// TIA Portal project "Elevator_V16" (V16)

(* hardware
DEVICE "S7-1200 station_1"  S7-1200 Station
   slot 0: "Rack_0"  S7-1200 Rack  Rack  V1.0
   slot 1: "PLC_1"  CPU 1217C DC/DC/DC  6ES7 217-1AG40-0XB0  V4.2
DEVICE "HMI_1"  KTP700 Basic PN
   slot 0: "KTP700 Basic PN"  KTP700 Basic PN  6AV2 123-2GB03-0AX0  14.0.1.0
   slot 1: "HMI_RT_1"  KTP700 Basic PN  6AV2 123-2GB03-0AX0  14.0.1.0
   slot 5: "HMI_1.IE_CP_1"  PROFINET Interface  14.0.1.0
      slot 1: "PROFINET Interface_1"  PROFINET Interface
         slot 1: "Port_1"  Port
*)

// ===== PLC "PLC_1"  CPU 1217C DC/DC/DC =====

VAR_GLOBAL   // PLC tag table "Default tag table"
   "Tag_1" AT %M20.0 : Bool;
END_VAR

DATA_BLOCK "DB_Main"   // DB1
{ S7_Optimized_Access := 'TRUE' }
VERSION : 0.1
   VAR
      Floor1 : Struct
         Request_PB : Bool;
         OpenDoor : Bool;
         OpenDoor_Timer : TON_TIME;
         OneShot_1 : Bool;
      END_STRUCT;
      Floor2 : Struct
         Request_PB : Bool;
         OpenDoor : Bool;
         OpenDoor_Timer : TON_TIME;
         OneShot_1 : Bool;
      END_STRUCT;
      Floor3 : Struct
         Request_PB : Bool;
         OpenDoor : Bool;
         OpenDoor_Timer : TON_TIME;
         OneShot_1 : Bool;
      END_STRUCT;
      Elevator : Struct
         Floor1_PB : Bool;
         Floor2_PB : Bool;
         Floor3_PB : Bool;
         Floor1_Scheduled : Bool;
         Floor2_Scheduled : Bool;
         Floor3_Scheduled : Bool;
         At_Floor1 : Bool;
         At_Floor2 : Bool;
         At_Floor3 : Bool;
         CurrentFloor : Int;
         NextFloorToService : Int;
         Motor_CW : Bool;
         Motor_CCW : Bool;
         GoingUp_Timer_1 : TON_TIME;
         GoingUp_Timer_2 : TON_TIME;
         GoingDown_Timer1 : TON_TIME;
         GoingDown_Timer2 : TON_TIME;
         OneShot_1 : Bool;
         OneShot_2 : Bool;
      END_STRUCT;
   END_VAR
BEGIN
END_DATA_BLOCK

ORGANIZATION_BLOCK "Main"   // OB1, LAD, ProgramCycle
TITLE = "Main Program Sweep (Cycle)"
{ S7_Optimized_Access := 'TRUE' }
VERSION : 0.1
   VAR_INPUT
      Initial_Call : Bool;   // Initial call of this OB
      Remanence : Bool;   // =True, if remanent data are available
   END_VAR
   VAR_TEMP   // added for the SCL form of the ladder/FBD networks
      _w1 : Bool;
      _w2 : Bool;
      _w3 : Bool;
      _w4 : Bool;
      _w5 : Bool;
      _w6 : Bool;
   END_VAR
BEGIN

REGION Network 1: Mange Scheduled Floors
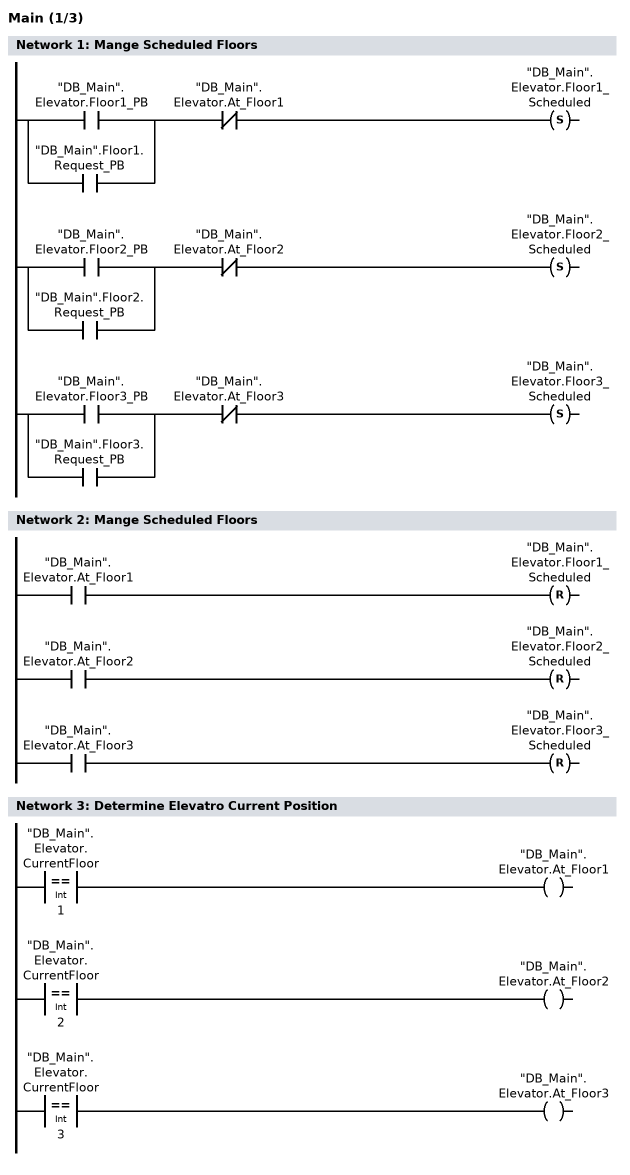
   RUNG wire#powerrail
      Contact( "DB_Main".Elevator.Floor1_PB )
      wire#w1
      I_Contact( "DB_Main".Elevator.At_Floor1 )
      S_Coil( "DB_Main".Elevator.Floor1_Scheduled )
   END_RUNG
   RUNG wire#powerrail
      Contact( "DB_Main".Floor1.Request_PB )
   END_RUNG wire#w1
   RUNG wire#powerrail
      Contact( "DB_Main".Elevator.Floor2_PB )
      wire#w2
      I_Contact( "DB_Main".Elevator.At_Floor2 )
      S_Coil( "DB_Main".Elevator.Floor2_Scheduled )
   END_RUNG
   RUNG wire#powerrail
      Contact( "DB_Main".Floor2.Request_PB )
   END_RUNG wire#w2
   RUNG wire#powerrail
      Contact( "DB_Main".Elevator.Floor3_PB )
      wire#w3
      I_Contact( "DB_Main".Elevator.At_Floor3 )
      S_Coil( "DB_Main".Elevator.Floor3_Scheduled )
   END_RUNG
   RUNG wire#powerrail
      Contact( "DB_Main".Floor3.Request_PB )
   END_RUNG wire#w3
   // the same network as SCL:
   IF ("DB_Main".Elevator.Floor1_PB OR "DB_Main".Floor1.Request_PB) AND NOT "DB_Main".Elevator.At_Floor1 THEN
       "DB_Main".Elevator.Floor1_Scheduled := TRUE;
   END_IF;
   IF ("DB_Main".Elevator.Floor2_PB OR "DB_Main".Floor2.Request_PB) AND NOT "DB_Main".Elevator.At_Floor2 THEN
       "DB_Main".Elevator.Floor2_Scheduled := TRUE;
   END_IF;
   IF ("DB_Main".Elevator.Floor3_PB OR "DB_Main".Floor3.Request_PB) AND NOT "DB_Main".Elevator.At_Floor3 THEN
       "DB_Main".Elevator.Floor3_Scheduled := TRUE;
   END_IF;
END_REGION

REGION Network 2: Mange Scheduled Floors
   RUNG wire#powerrail
      Contact( "DB_Main".Elevator.At_Floor1 )
      R_Coil( "DB_Main".Elevator.Floor1_Scheduled )
   END_RUNG
   RUNG wire#powerrail
      Contact( "DB_Main".Elevator.At_Floor2 )
      R_Coil( "DB_Main".Elevator.Floor2_Scheduled )
   END_RUNG
   RUNG wire#powerrail
      Contact( "DB_Main".Elevator.At_Floor3 )
      R_Coil( "DB_Main".Elevator.Floor3_Scheduled )
   END_RUNG
   // the same network as SCL:
   IF "DB_Main".Elevator.At_Floor1 THEN "DB_Main".Elevator.Floor1_Scheduled := FALSE; END_IF;
   IF "DB_Main".Elevator.At_Floor2 THEN "DB_Main".Elevator.Floor2_Scheduled := FALSE; END_IF;
   IF "DB_Main".Elevator.At_Floor3 THEN "DB_Main".Elevator.Floor3_Scheduled := FALSE; END_IF;
END_REGION

REGION Network 3: Determine Elevatro Current Position
   RUNG wire#powerrail
      { S7_Templates := "SrcType := Int" } EQ_Contact(in1 := "DB_Main".Elevator.CurrentFloor, in2 := 1)
      Coil( "DB_Main".Elevator.At_Floor1 )
   END_RUNG
   RUNG wire#powerrail
      { S7_Templates := "SrcType := Int" } EQ_Contact(in1 := "DB_Main".Elevator.CurrentFloor, in2 := 2)
      Coil( "DB_Main".Elevator.At_Floor2 )
   END_RUNG
   RUNG wire#powerrail
      { S7_Templates := "SrcType := Int" } EQ_Contact(in1 := "DB_Main".Elevator.CurrentFloor, in2 := 3)
      Coil( "DB_Main".Elevator.At_Floor3 )
   END_RUNG
   // the same network as SCL:
   "DB_Main".Elevator.At_Floor1 := "DB_Main".Elevator.CurrentFloor = 1;
   "DB_Main".Elevator.At_Floor2 := "DB_Main".Elevator.CurrentFloor = 2;
   "DB_Main".Elevator.At_Floor3 := "DB_Main".Elevator.CurrentFloor = 3;
END_REGION

REGION Network 4: Determine Service Priorities
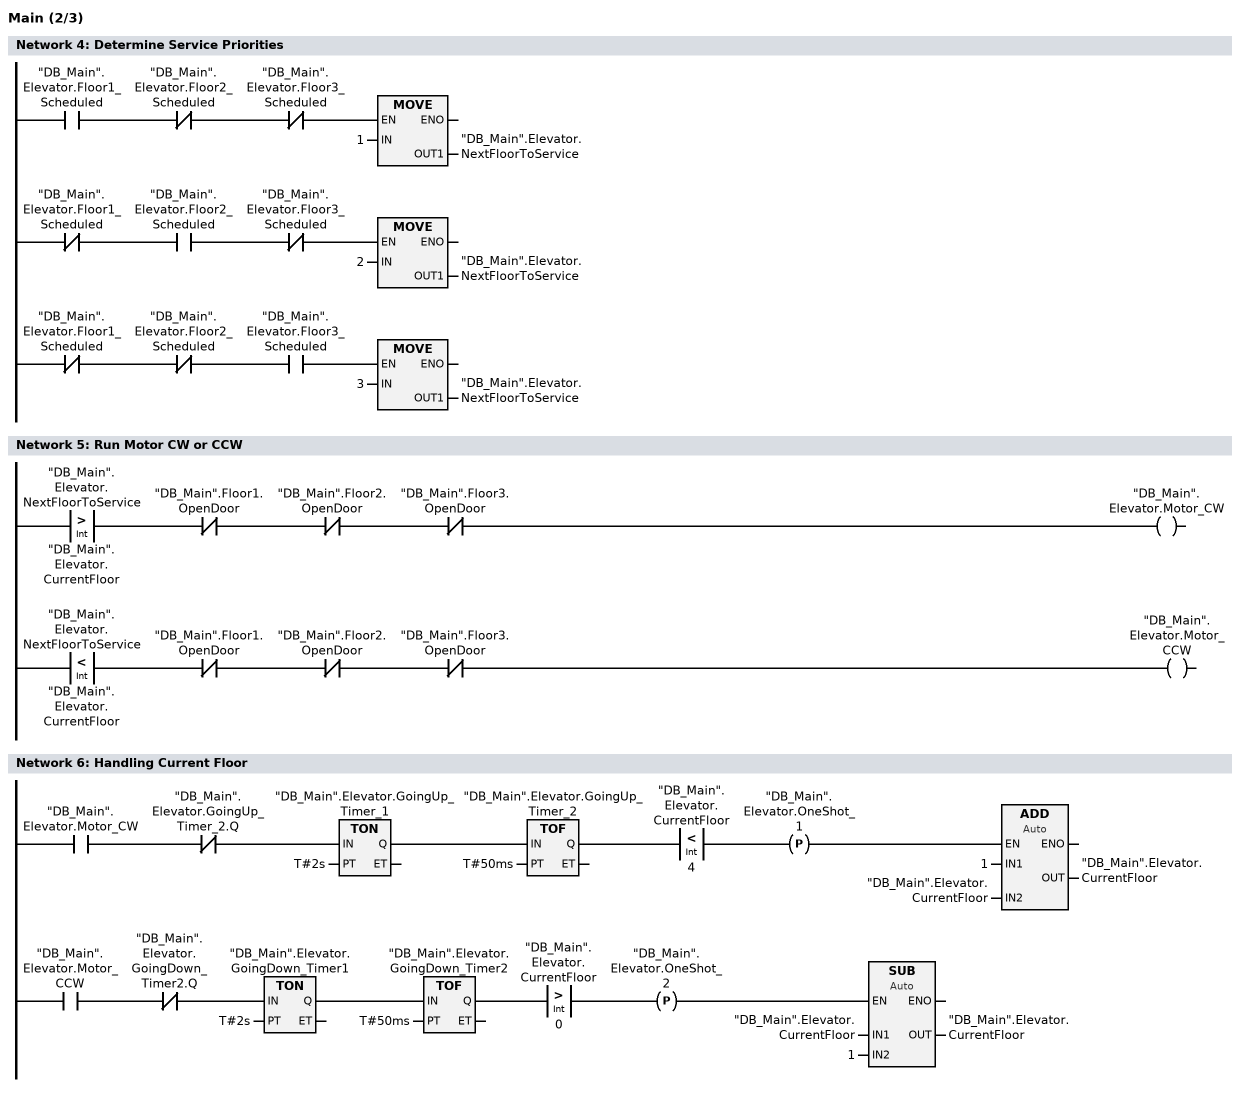
   RUNG wire#powerrail
      Contact( "DB_Main".Elevator.Floor1_Scheduled )
      I_Contact( "DB_Main".Elevator.Floor2_Scheduled )
      I_Contact( "DB_Main".Elevator.Floor3_Scheduled )
      Move(in := 1, out1 => "DB_Main".Elevator.NextFloorToService)
   END_RUNG
   RUNG wire#powerrail
      I_Contact( "DB_Main".Elevator.Floor1_Scheduled )
      Contact( "DB_Main".Elevator.Floor2_Scheduled )
      I_Contact( "DB_Main".Elevator.Floor3_Scheduled )
      Move(in := 2, out1 => "DB_Main".Elevator.NextFloorToService)
   END_RUNG
   RUNG wire#powerrail
      I_Contact( "DB_Main".Elevator.Floor1_Scheduled )
      I_Contact( "DB_Main".Elevator.Floor2_Scheduled )
      Contact( "DB_Main".Elevator.Floor3_Scheduled )
      Move(in := 3, out1 => "DB_Main".Elevator.NextFloorToService)
   END_RUNG
   // the same network as SCL:
   IF "DB_Main".Elevator.Floor1_Scheduled AND NOT "DB_Main".Elevator.Floor2_Scheduled AND NOT "DB_Main".Elevator.Floor3_Scheduled THEN
       "DB_Main".Elevator.NextFloorToService := 1;
   END_IF;
   IF NOT "DB_Main".Elevator.Floor1_Scheduled AND "DB_Main".Elevator.Floor2_Scheduled AND NOT "DB_Main".Elevator.Floor3_Scheduled THEN
       "DB_Main".Elevator.NextFloorToService := 2;
   END_IF;
   IF NOT "DB_Main".Elevator.Floor1_Scheduled AND NOT "DB_Main".Elevator.Floor2_Scheduled AND "DB_Main".Elevator.Floor3_Scheduled THEN
       "DB_Main".Elevator.NextFloorToService := 3;
   END_IF;
END_REGION

REGION Network 5: Run Motor CW or CCW
   RUNG wire#powerrail
      { S7_Templates := "SrcType := Int" } GT_Contact(in1 := "DB_Main".Elevator.NextFloorToService, in2 := "DB_Main".Elevator.CurrentFloor)
      I_Contact( "DB_Main".Floor1.OpenDoor )
      I_Contact( "DB_Main".Floor2.OpenDoor )
      I_Contact( "DB_Main".Floor3.OpenDoor )
      Coil( "DB_Main".Elevator.Motor_CW )
   END_RUNG
   RUNG wire#powerrail
      { S7_Templates := "SrcType := Int" } LT_Contact(in1 := "DB_Main".Elevator.NextFloorToService, in2 := "DB_Main".Elevator.CurrentFloor)
      I_Contact( "DB_Main".Floor1.OpenDoor )
      I_Contact( "DB_Main".Floor2.OpenDoor )
      I_Contact( "DB_Main".Floor3.OpenDoor )
      Coil( "DB_Main".Elevator.Motor_CCW )
   END_RUNG
   // the same network as SCL:
   "DB_Main".Elevator.Motor_CW := ("DB_Main".Elevator.NextFloorToService > "DB_Main".Elevator.CurrentFloor) AND NOT "DB_Main".Floor1.OpenDoor AND NOT "DB_Main".Floor2.OpenDoor AND NOT "DB_Main".Floor3.OpenDoor;
   "DB_Main".Elevator.Motor_CCW := ("DB_Main".Elevator.NextFloorToService < "DB_Main".Elevator.CurrentFloor) AND NOT "DB_Main".Floor1.OpenDoor AND NOT "DB_Main".Floor2.OpenDoor AND NOT "DB_Main".Floor3.OpenDoor;
END_REGION

REGION Network 6: Handling Current Floor
   "DB_Main".Elevator.GoingUp_Timer_1.TON(IN := "DB_Main".Elevator.Motor_CW AND NOT "DB_Main".Elevator.GoingUp_Timer_2.Q,
                           PT := T#2s);
   "DB_Main".Elevator.GoingUp_Timer_2.TOF(IN := "DB_Main".Elevator.GoingUp_Timer_1.Q, PT := T#50ms);
   #_w1 := "DB_Main".Elevator.GoingUp_Timer_2.Q AND ("DB_Main".Elevator.CurrentFloor < 4);
   #_w2 := #_w1 AND NOT "DB_Main".Elevator.OneShot_1;   // rising edge
   "DB_Main".Elevator.OneShot_1 := #_w1;
   IF #_w2 THEN "DB_Main".Elevator.CurrentFloor := 1 + "DB_Main".Elevator.CurrentFloor; END_IF;
   "DB_Main".Elevator.GoingDown_Timer1.TON(IN := "DB_Main".Elevator.Motor_CCW AND NOT "DB_Main".Elevator.GoingDown_Timer2.Q,
                           PT := T#2s);
   "DB_Main".Elevator.GoingDown_Timer2.TOF(IN := "DB_Main".Elevator.GoingDown_Timer1.Q, PT := T#50ms);
   #_w3 := "DB_Main".Elevator.GoingDown_Timer2.Q AND ("DB_Main".Elevator.CurrentFloor > 0);
   #_w4 := #_w3 AND NOT "DB_Main".Elevator.OneShot_2;   // rising edge
   "DB_Main".Elevator.OneShot_2 := #_w3;
   IF #_w4 THEN "DB_Main".Elevator.CurrentFloor := "DB_Main".Elevator.CurrentFloor - 1; END_IF;
END_REGION

REGION Network 7: Door Handling
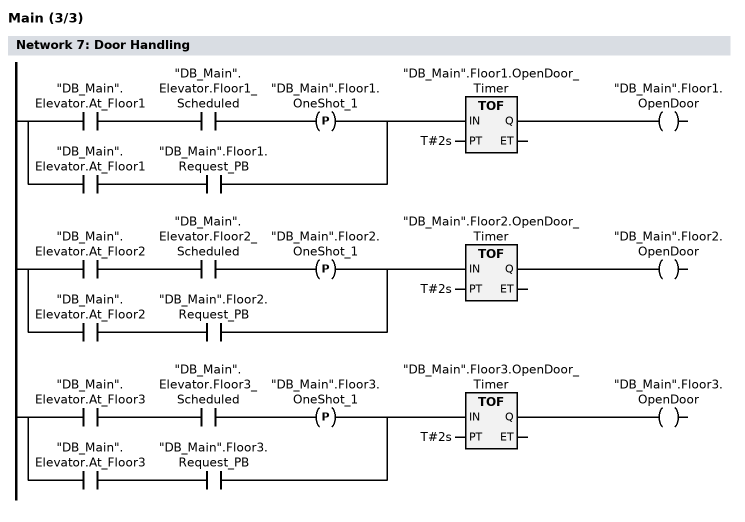
   #_w1 := "DB_Main".Elevator.At_Floor1 AND "DB_Main".Elevator.Floor1_Scheduled;
   #_w2 := #_w1 AND NOT "DB_Main".Floor1.OneShot_1;   // rising edge
   "DB_Main".Floor1.OneShot_1 := #_w1;
   "DB_Main".Floor1.OpenDoor_Timer.TOF(IN := #_w2 OR ("DB_Main".Elevator.At_Floor1 AND "DB_Main".Floor1.Request_PB),
                           PT := T#2s);
   "DB_Main".Floor1.OpenDoor := "DB_Main".Floor1.OpenDoor_Timer.Q;
   #_w3 := "DB_Main".Elevator.At_Floor2 AND "DB_Main".Elevator.Floor2_Scheduled;
   #_w4 := #_w3 AND NOT "DB_Main".Floor2.OneShot_1;   // rising edge
   "DB_Main".Floor2.OneShot_1 := #_w3;
   "DB_Main".Floor2.OpenDoor_Timer.TOF(IN := #_w4 OR ("DB_Main".Elevator.At_Floor2 AND "DB_Main".Floor2.Request_PB),
                           PT := T#2s);
   "DB_Main".Floor2.OpenDoor := "DB_Main".Floor2.OpenDoor_Timer.Q;
   #_w5 := "DB_Main".Elevator.At_Floor3 AND "DB_Main".Elevator.Floor3_Scheduled;
   #_w6 := #_w5 AND NOT "DB_Main".Floor3.OneShot_1;   // rising edge
   "DB_Main".Floor3.OneShot_1 := #_w5;
   "DB_Main".Floor3.OpenDoor_Timer.TOF(IN := #_w6 OR ("DB_Main".Elevator.At_Floor3 AND "DB_Main".Floor3.Request_PB),
                           PT := T#2s);
   "DB_Main".Floor3.OpenDoor := "DB_Main".Floor3.OpenDoor_Timer.Q;
END_REGION
END_ORGANIZATION_BLOCK

(* ===== HMI "HMI_RT_1" =====
system functions are stored by id; their names below are inferred from use
connection "HMI_Connection_1": ETHERNET, SMART_S7_1200_OMS

HMI tags "Default tag table"
   "DB_Main_Floor1_Request_PB" : Bool = PLC DB_Main.Floor1.Request_PB, 1 s
   "DB_Main_Floor1_OpenDoor" : Bool = PLC DB_Main.Floor1.OpenDoor, 1 s
   "DB_Main_Floor1_OpenDoor_Timer_PT" : Time = PLC DB_Main.Floor1.OpenDoor_Timer.PT, 1 s
   "DB_Main_Floor1_OpenDoor_Timer_ET" : Time = PLC DB_Main.Floor1.OpenDoor_Timer.ET, 1 s
   "DB_Main_Floor1_OpenDoor_Timer_IN" : Bool = PLC DB_Main.Floor1.OpenDoor_Timer.IN, 1 s
   "DB_Main_Floor1_OpenDoor_Timer_Q" : Bool = PLC DB_Main.Floor1.OpenDoor_Timer.Q, 1 s
   "DB_Main_Floor1_OneShot_1" : Bool = PLC DB_Main.Floor1.OneShot_1, 1 s
   "DB_Main_Floor2_Request_PB" : Bool = PLC DB_Main.Floor2.Request_PB, 1 s
   "DB_Main_Floor2_OpenDoor" : Bool = PLC DB_Main.Floor2.OpenDoor, 1 s
   "DB_Main_Floor2_OpenDoor_Timer_PT" : Time = PLC DB_Main.Floor2.OpenDoor_Timer.PT, 1 s
   "DB_Main_Floor2_OpenDoor_Timer_ET" : Time = PLC DB_Main.Floor2.OpenDoor_Timer.ET, 1 s
   "DB_Main_Floor2_OpenDoor_Timer_IN" : Bool = PLC DB_Main.Floor2.OpenDoor_Timer.IN, 1 s
   "DB_Main_Floor2_OpenDoor_Timer_Q" : Bool = PLC DB_Main.Floor2.OpenDoor_Timer.Q, 1 s
   "DB_Main_Floor2_OneShot_1" : Bool = PLC DB_Main.Floor2.OneShot_1, 1 s
   "DB_Main_Floor3_Request_PB" : Bool = PLC DB_Main.Floor3.Request_PB, 1 s
   "DB_Main_Floor3_OpenDoor" : Bool = PLC DB_Main.Floor3.OpenDoor, 1 s
   "DB_Main_Floor3_OpenDoor_Timer_PT" : Time = PLC DB_Main.Floor3.OpenDoor_Timer.PT, 1 s
   "DB_Main_Floor3_OpenDoor_Timer_ET" : Time = PLC DB_Main.Floor3.OpenDoor_Timer.ET, 1 s
   "DB_Main_Floor3_OpenDoor_Timer_IN" : Bool = PLC DB_Main.Floor3.OpenDoor_Timer.IN, 1 s
   "DB_Main_Floor3_OpenDoor_Timer_Q" : Bool = PLC DB_Main.Floor3.OpenDoor_Timer.Q, 1 s
   "DB_Main_Floor3_OneShot_1" : Bool = PLC DB_Main.Floor3.OneShot_1, 1 s
   "DB_Main_Elevator_Floor1_PB" : Bool = PLC DB_Main.Elevator.Floor1_PB, 1 s
   "DB_Main_Elevator_Floor2_PB" : Bool = PLC DB_Main.Elevator.Floor2_PB, 1 s
   "DB_Main_Elevator_Floor3_PB" : Bool = PLC DB_Main.Elevator.Floor3_PB, 1 s
   "DB_Main_Elevator_Floor1_Scheduled" : Bool = PLC DB_Main.Elevator.Floor1_Scheduled, 1 s
   "DB_Main_Elevator_Floor2_Scheduled" : Bool = PLC DB_Main.Elevator.Floor2_Scheduled, 1 s
   "DB_Main_Elevator_Floor3_Scheduled" : Bool = PLC DB_Main.Elevator.Floor3_Scheduled, 1 s
   "DB_Main_Elevator_At_Floor1" : Bool = PLC DB_Main.Elevator.At_Floor1, 1 s
   "DB_Main_Elevator_At_Floor2" : Bool = PLC DB_Main.Elevator.At_Floor2, 1 s
   "DB_Main_Elevator_At_Floor3" : Bool = PLC DB_Main.Elevator.At_Floor3, 1 s
   "DB_Main_Elevator_CurrentFloor" : Int = PLC DB_Main.Elevator.CurrentFloor, 1 s
   "DB_Main_Elevator_NextFloorToService" : Int = PLC DB_Main.Elevator.NextFloorToService, 1 s
   "DB_Main_Elevator_Motor_CW" : Bool = PLC DB_Main.Elevator.Motor_CW, 1 s
   "DB_Main_Elevator_Motor_CCW" : Bool = PLC DB_Main.Elevator.Motor_CCW, 1 s
   "DB_Main_Elevator_GoingUp_Timer_1_PT" : Time = PLC DB_Main.Elevator.GoingUp_Timer_1.PT, 1 s
   "DB_Main_Elevator_GoingUp_Timer_1_ET" : Time = PLC DB_Main.Elevator.GoingUp_Timer_1.ET, 1 s
   "DB_Main_Elevator_GoingUp_Timer_1_IN" : Bool = PLC DB_Main.Elevator.GoingUp_Timer_1.IN, 1 s
   "DB_Main_Elevator_GoingUp_Timer_1_Q" : Bool = PLC DB_Main.Elevator.GoingUp_Timer_1.Q, 1 s
   "DB_Main_Elevator_GoingUp_Timer_2_PT" : Time = PLC DB_Main.Elevator.GoingUp_Timer_2.PT, 1 s
   "DB_Main_Elevator_GoingUp_Timer_2_ET" : Time = PLC DB_Main.Elevator.GoingUp_Timer_2.ET, 1 s
   "DB_Main_Elevator_GoingUp_Timer_2_IN" : Bool = PLC DB_Main.Elevator.GoingUp_Timer_2.IN, 1 s
   "DB_Main_Elevator_GoingUp_Timer_2_Q" : Bool = PLC DB_Main.Elevator.GoingUp_Timer_2.Q, 1 s
   "DB_Main_Elevator_GoingDown_Timer1_PT" : Time = PLC DB_Main.Elevator.GoingDown_Timer1.PT, 1 s
   "DB_Main_Elevator_GoingDown_Timer1_ET" : Time = PLC DB_Main.Elevator.GoingDown_Timer1.ET, 1 s
   "DB_Main_Elevator_GoingDown_Timer1_IN" : Bool = PLC DB_Main.Elevator.GoingDown_Timer1.IN, 1 s
   "DB_Main_Elevator_GoingDown_Timer1_Q" : Bool = PLC DB_Main.Elevator.GoingDown_Timer1.Q, 1 s
   "DB_Main_Elevator_GoingDown_Timer2_PT" : Time = PLC DB_Main.Elevator.GoingDown_Timer2.PT, 1 s
   "DB_Main_Elevator_GoingDown_Timer2_ET" : Time = PLC DB_Main.Elevator.GoingDown_Timer2.ET, 1 s
   "DB_Main_Elevator_GoingDown_Timer2_IN" : Bool = PLC DB_Main.Elevator.GoingDown_Timer2.IN, 1 s
   "DB_Main_Elevator_GoingDown_Timer2_Q" : Bool = PLC DB_Main.Elevator.GoingDown_Timer2.Q, 1 s
   "DB_Main_Elevator_OneShot_1" : Bool = PLC DB_Main.Elevator.OneShot_1, 1 s
   "DB_Main_Elevator_OneShot_2" : Bool = PLC DB_Main.Elevator.OneShot_2, 1 s

screen "Elevator_Control" 800x480
   Button "Button_1" at 320,143 size 23x23; TextOff 'Text'; PictureOff "Down_Arrow"
      on Release: ResetBit("DB_Main_Floor3_Request_PB")
      on Press: SetBit("DB_Main_Floor3_Request_PB")
   TextField "Text field_4" at 320,49 size 113x23; Text 'Current Floor'
   IOField "I/O field_1" at 439,47 size 56x27; FormatPattern 99
      ProcessValue <- "DB_Main_Elevator_CurrentFloor"
   Button "Button_2" at 320,263 size 23x23; TextOff 'Text'; PictureOff "UPDOWN"
      on Press: SetBit("DB_Main_Floor2_Request_PB")
      on Release: ResetBit("DB_Main_Floor2_Request_PB")
   Button "Button_9" at 320,383 size 23x23; TextOff 'Text'; PictureOff "Up_Arrow"
      on Press: SetBit("DB_Main_Floor1_Request_PB")
      on Release: ResetBit("DB_Main_Floor1_Request_PB")
   Rectangle "Rectangle_2" at 470,232 size 39x85
      Visibility <- "DB_Main_Elevator_At_Floor2"
   Rectangle "Rectangle_6" at 393,239 size 32x73
      Visibility <- "DB_Main_Floor2_OpenDoor"
   Rectangle "Rectangle_7" at 426,239 size 32x73
      Visibility <- "DB_Main_Floor2_OpenDoor"
   Rectangle "Rectangle_8" at 393,239 size 9x73
      Visibility <- "DB_Main_Floor2_OpenDoor"
   Rectangle "Rectangle_9" at 450,239 size 9x73
      Visibility <- "DB_Main_Floor2_OpenDoor"
   Button "Button_3" at 476,236 size 28x25; TextOff '3'
      on Release: ResetBit("DB_Main_Elevator_Floor3_PB")
      Visibility <- "DB_Main_Elevator_At_Floor2"
      on Press: SetBit("DB_Main_Elevator_Floor3_PB")
      Appearance <- "DB_Main_Elevator_Floor3_Scheduled"
   Button "Button_7" at 476,262 size 28x25; TextOff '2'
      on Release: ResetBit("DB_Main_Elevator_Floor2_PB")
      on Press: SetBit("DB_Main_Elevator_Floor2_PB")
      Visibility <- "DB_Main_Elevator_At_Floor2"
      Appearance <- "DB_Main_Elevator_Floor2_Scheduled"
   Button "Button_8" at 476,288 size 28x25; TextOff '1'
      on Release: ResetBit("DB_Main_Elevator_Floor1_PB")
      on Press: SetBit("DB_Main_Elevator_Floor1_PB")
      Visibility <- "DB_Main_Elevator_At_Floor2"
      Appearance <- "DB_Main_Elevator_Floor1_Scheduled"
   Rectangle "Rectangle_13" at 470,352 size 39x85
      Visibility <- "DB_Main_Elevator_At_Floor1"
   Rectangle "Rectangle_14" at 393,359 size 32x73
      Visibility <- "DB_Main_Floor1_OpenDoor"
   Rectangle "Rectangle_15" at 426,359 size 32x73
      Visibility <- "DB_Main_Floor1_OpenDoor"
   Rectangle "Rectangle_18" at 393,359 size 9x73
      Visibility <- "DB_Main_Floor1_OpenDoor"
   Rectangle "Rectangle_19" at 450,359 size 9x73
      Visibility <- "DB_Main_Floor1_OpenDoor"
   Button "Button_10" at 476,356 size 28x25; TextOff '3'
      on Release: ResetBit("DB_Main_Elevator_Floor3_PB")
      Visibility <- "DB_Main_Elevator_At_Floor1"
      on Press: SetBit("DB_Main_Elevator_Floor3_PB")
      Appearance <- "DB_Main_Elevator_Floor3_Scheduled"
   Button "Button_11" at 476,382 size 28x25; TextOff '2'
      on Release: ResetBit("DB_Main_Elevator_Floor2_PB")
      on Press: SetBit("DB_Main_Elevator_Floor2_PB")
      Visibility <- "DB_Main_Elevator_At_Floor1"
      Appearance <- "DB_Main_Elevator_Floor2_Scheduled"
   Button "Button_12" at 476,408 size 28x25; TextOff '1'
      on Release: ResetBit("DB_Main_Elevator_Floor1_PB")
      on Press: SetBit("DB_Main_Elevator_Floor1_PB")
      Visibility <- "DB_Main_Elevator_At_Floor1"
      Appearance <- "DB_Main_Elevator_Floor1_Scheduled"
   Rectangle "Rectangle_17" at 470,112 size 39x85
      Visibility <- "DB_Main_Elevator_At_Floor3"
   Rectangle "Rectangle_5" at 393,119 size 32x73
      Visibility <- "DB_Main_Floor3_OpenDoor"
   Rectangle "Rectangle_4" at 426,119 size 32x73
      Visibility <- "DB_Main_Floor3_OpenDoor"
   Rectangle "Rectangle_10" at 393,119 size 9x73
      Visibility <- "DB_Main_Floor3_OpenDoor"
   Rectangle "Rectangle_11" at 450,119 size 9x73
      Visibility <- "DB_Main_Floor3_OpenDoor"
   Button "Button_4" at 476,116 size 28x25; TextOff '3'
      on Release: ResetBit("DB_Main_Elevator_Floor3_PB")
      on Press: SetBit("DB_Main_Elevator_Floor3_PB")
      Visibility <- "DB_Main_Elevator_At_Floor3"
      Appearance <- "DB_Main_Elevator_Floor3_Scheduled"
   Button "Button_5" at 476,142 size 28x25; TextOff '2'
      on Press: SetBit("DB_Main_Elevator_Floor2_PB")
      on Release: ResetBit("DB_Main_Elevator_Floor2_PB")
      Visibility <- "DB_Main_Elevator_At_Floor3"
      Appearance <- "DB_Main_Elevator_Floor2_Scheduled"
   Button "Button_6" at 476,168 size 28x25; TextOff '1'
      on Press: SetBit("DB_Main_Elevator_Floor1_PB")
      on Release: ResetBit("DB_Main_Elevator_Floor1_PB")
      Visibility <- "DB_Main_Elevator_At_Floor3"
      Appearance <- "DB_Main_Elevator_Floor1_Scheduled"
   TextField "Text field_1" at 33,25 size 203x28; Text '3 FLOOR ELEVATOR'
   Rectangle "Rectangle_21" at 320,143 size 23x23
      Visibility <- "DB_Main_Elevator_Floor3_Scheduled"
   Rectangle "Rectangle_22" at 320,263 size 23x23
      Visibility <- "DB_Main_Elevator_Floor2_Scheduled"
   Rectangle "Rectangle_23" at 320,383 size 23x23
      Visibility <- "DB_Main_Elevator_Floor1_Scheduled"
*)